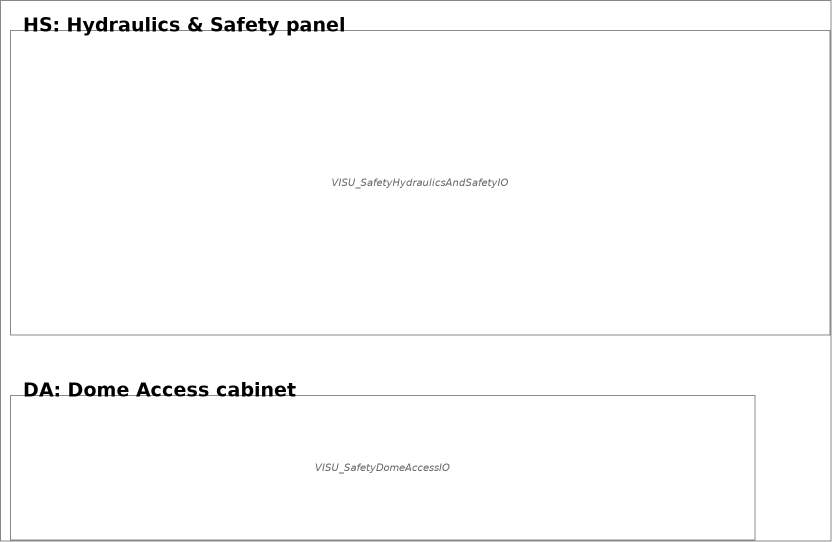
VISUALIZATION VISU_SafetyIO  // 832x542
VAR_IN_OUT
	ref : SafetyIO;
    widget : SafetyIOWidget;
END_VAR
    Frame (10,30 820x305)
        shows VISU_SafetyHydraulicsAndSafetyIO(ref := ref.parts.hydraulicsAndSafety, widget := widget.hydraulicsAndSafety)
        shows VISU_SafetyDomeAccessIO()
    Frame (10,395 745x145)
        shows VISU_SafetyDomeAccessIO(ref := ref.parts.domeAccess, widget := widget.domeAccess)
        shows VISU_SafetyDomeAccessIO()
    Label (20,10 350x30), "HS: Hydraulics & Safety panel"
    Label (20,375 350x30), "DA: Dome Access cabinet"
END_VISUALIZATION

(* stored: Version 1.1.0.1, ProductVersion 3.1.4019.2
   Visu VISU_SafetyIO: Id {4978f974-4464-46da-8445-997ee3cca1ac} *)
